// TwinCAT 3 PLC project PlcElevator
// ProgramVersion: 3.1.4024.0
// libraries:
//   Tc2_Standard, * (Beckhoff Automation GmbH)
//   Tc2_System, * (Beckhoff Automation GmbH)
//   Tc3_Module, * (Beckhoff Automation GmbH)
// project tree:
//   DUTs/ E_DoorState.TcDUT
//   GVLs/ GVL_HMI.TcGVL
//   / PlcTask.TcTTO
//   POUs/ FB_Dispatcher.TcPOU, FB_ElevatorCar.TcPOU, I_ElevatorCar.TcPOU, MAIN.TcPOU
// real-time tasks:
//   TASK PlcTask: cycle T#10ms, priority 20, ADS port 350

CONFIGURATION PlcElevator
    RESOURCE PLC ON TwinCAT3
        TASK PlcTask(INTERVAL := T#10ms, PRIORITY := 20);
        PROGRAM MAIN WITH PlcTask : MAIN;
    END_RESOURCE
END_CONFIGURATION

// ---- DUTs/E_DoorState.TcDUT
{attribute 'qualified_only'}
{attribute 'strict'}
TYPE E_DoorState :
(
	CLOSED := 0,
	OPENING := 1,
	OPEN := 2,
	CLOSING := 3
) INT;
END_TYPE

// ---- GVLs/GVL_HMI.TcGVL
{attribute 'qualified_only'}
VAR_GLOBAL
	bFloorCallsOutside : ARRAY[1..10] OF BOOL; // HMI Landing Call Buttons
	bCabinCallsInside  : ARRAY[1..10] OF BOOL; // HMI Internal Cabin Buttons
	bHmiObstruction    : BOOL;                // HMI Door Obstruction Toggle
	
	// Status Feedbacks for HMI Animation
	rfHmiCabinPosition : LREAL := 1.0;        // Continuous position (1.0 to 10.0)
	nHmiCurrentFloor   : INT := 1;            // Discrete Current Floor
	eHmiDoorState      : INT;                 // Casted E_DoorState for HMI binding
	bHmiMovingUp       : BOOL;                // Cabin is moving up
	bHmiMovingDown     : BOOL;                // Cabin is moving down
	nHmiTargetFloor    : INT;                 // Current Target Floor
END_VAR

// ---- POUs/I_ElevatorCar.TcPOU
INTERFACE I_ElevatorCar

PROPERTY CurrentFloor : INT
GET
END_GET
END_PROPERTY

PROPERTY DoorState : E_DoorState
GET
END_GET
END_PROPERTY

PROPERTY IsBusy : BOOL
GET
END_GET
END_PROPERTY

METHOD MoveToFloor : BOOL
VAR_INPUT
	nFloor : INT;
END_VAR
END_METHOD

METHOD OpenDoors : BOOL
END_METHOD

PROPERTY Position : LREAL
GET
END_GET
END_PROPERTY

END_INTERFACE

// ---- POUs/MAIN.TcPOU
PROGRAM MAIN
VAR
	fbCar : FB_ElevatorCar;
	fbDispatcher : FB_Dispatcher;

	// Automated Test Harness
	bRunTestCases : BOOL := FALSE;
	nTestStep : INT := 0;
	iTest : INT;
END_VAR

// Execute the physical elevator cabin simulation and door state machine
fbCar();

// Execute dispatcher to run SCAN sorting algorithm
fbDispatcher.Update(fbCar);

// Bind local state feedbacks to GVL_HMI for HMI animation and telemetry
GVL_HMI.rfHmiCabinPosition := fbCar.Position;
GVL_HMI.nHmiCurrentFloor   := fbCar.CurrentFloor;
GVL_HMI.eHmiDoorState      := TO_INT(fbCar.DoorState);
GVL_HMI.bHmiMovingUp       := fbDispatcher.bMovingUp;
GVL_HMI.bHmiMovingDown     := fbDispatcher.bMovingDown;
GVL_HMI.nHmiTargetFloor    := fbDispatcher.nTargetFloor;

// Automated Test Runner (Self-Verification)
IF bRunTestCases THEN
	CASE nTestStep OF
		0: // Step 0: Initialize test, clear all calls, reset cabin to floor 1
			FOR iTest := 1 TO 10 DO
				GVL_HMI.bFloorCallsOutside[iTest] := FALSE;
				GVL_HMI.bCabinCallsInside[iTest] := FALSE;
			END_FOR
			fbCar.MoveToFloor(1);
			nTestStep := 1;
			
		1: // Step 1: Wait for cabin to reach floor 1 and become idle
			IF fbCar.CurrentFloor = 1 AND NOT fbCar.IsBusy THEN
				// Place calls at floor 10 and floor 5
				GVL_HMI.bFloorCallsOutside[10] := TRUE;
				GVL_HMI.bFloorCallsOutside[5]  := TRUE;
				nTestStep := 2;
			END_IF
			
		2: // Step 2: Verify it stops at Floor 5 on the way up and clears call
			IF fbCar.CurrentFloor = 5 AND fbCar.DoorState = E_DoorState.OPEN THEN
				IF NOT GVL_HMI.bFloorCallsOutside[5] THEN
					// Floor 5 stop verified and call cleared successfully!
					nTestStep := 3;
				END_IF
			END_IF
			
		3: // Step 3: Wait for cabin to reach Floor 10 and clear call
			IF fbCar.CurrentFloor = 10 AND fbCar.DoorState = E_DoorState.OPEN THEN
				IF NOT GVL_HMI.bFloorCallsOutside[10] THEN
					// Floor 10 stop verified and call cleared successfully!
					// Test passed!
					bRunTestCases := FALSE;
					nTestStep := 0;
				END_IF
			END_IF
	END_CASE
END_IF

END_PROGRAM

// ---- POUs/FB_ElevatorCar.TcPOU
FUNCTION_BLOCK FB_ElevatorCar IMPLEMENTS I_ElevatorCar
VAR
	rfPosition : LREAL := 1.0;
	nTargetFloor : INT := 1;
	eDoorState : E_DoorState := E_DoorState.CLOSED;
	bMoving : BOOL := FALSE;
	bObstruction : BOOL := FALSE;
	bTriggerDoorOpen : BOOL := FALSE;

	fbDoorDwellTimer : TON;
	fbOpeningTimer : TON;
	fbClosingTimer : TON;
END_VAR

// Synchronize door obstruction from external HMI/safety input
bObstruction := GVL_HMI.bHmiObstruction;

// Door State Machine
CASE eDoorState OF
	E_DoorState.CLOSED:
		fbOpeningTimer(IN := FALSE);
		fbDoorDwellTimer(IN := FALSE);
		fbClosingTimer(IN := FALSE);
		
		IF bTriggerDoorOpen THEN
			bTriggerDoorOpen := FALSE;
			eDoorState := E_DoorState.OPENING;
		END_IF
		
	E_DoorState.OPENING:
		fbOpeningTimer(IN := TRUE, PT := T#1S); // 1s opening time
		IF fbOpeningTimer.Q THEN
			fbOpeningTimer(IN := FALSE);
			eDoorState := E_DoorState.OPEN;
		END_IF
		
	E_DoorState.OPEN:
		fbDoorDwellTimer(IN := NOT bObstruction, PT := T#3S); // 3s dwell timer
		IF fbDoorDwellTimer.Q THEN
			fbDoorDwellTimer(IN := FALSE);
			eDoorState := E_DoorState.CLOSING;
		END_IF
		
	E_DoorState.CLOSING:
		fbClosingTimer(IN := TRUE, PT := T#1S); // 1s closing time
		
		IF bObstruction THEN
			// Light Curtain obstruction: instantly reverse to OPENING
			fbClosingTimer(IN := FALSE);
			eDoorState := E_DoorState.OPENING;
		ELSIF fbClosingTimer.Q THEN
			fbClosingTimer(IN := FALSE);
			eDoorState := E_DoorState.CLOSED;
		END_IF
END_CASE

// Cabin Movement Logic (Safety Interlock)
IF eDoorState = E_DoorState.CLOSED THEN
	IF rfPosition < INT_TO_LREAL(nTargetFloor) THEN
		bMoving := TRUE;
		rfPosition := rfPosition + 0.02;
		IF rfPosition >= INT_TO_LREAL(nTargetFloor) THEN
			rfPosition := INT_TO_LREAL(nTargetFloor);
			bMoving := FALSE;
			bTriggerDoorOpen := TRUE; // Auto-open doors upon arrival
		END_IF
	ELSIF rfPosition > INT_TO_LREAL(nTargetFloor) THEN
		bMoving := TRUE;
		rfPosition := rfPosition - 0.02;
		IF rfPosition <= INT_TO_LREAL(nTargetFloor) THEN
			rfPosition := INT_TO_LREAL(nTargetFloor);
			bMoving := FALSE;
			bTriggerDoorOpen := TRUE; // Auto-open doors upon arrival
		END_IF
	ELSE
		bMoving := FALSE;
	END_IF
ELSE
	// Door is NOT closed - safety interlock: cabin CANNOT move
	bMoving := FALSE;
END_IF

METHOD MoveToFloor : BOOL
VAR_INPUT
	nFloor : INT;
END_VAR
IF nFloor >= 1 AND nFloor <= 10 AND eDoorState = E_DoorState.CLOSED THEN
	nTargetFloor := nFloor;
	MoveToFloor := TRUE;
ELSE
	MoveToFloor := FALSE;
END_IF
END_METHOD

METHOD OpenDoors : BOOL
IF NOT bMoving AND eDoorState = E_DoorState.CLOSED THEN
	bTriggerDoorOpen := TRUE;
	OpenDoors := TRUE;
ELSE
	OpenDoors := FALSE;
END_IF
END_METHOD

PROPERTY CurrentFloor : INT
GET
CurrentFloor := LREAL_TO_INT(rfPosition);
END_GET
END_PROPERTY

PROPERTY DoorState : E_DoorState
GET
DoorState := eDoorState;
END_GET
END_PROPERTY

PROPERTY IsBusy : BOOL
GET
IsBusy := bMoving OR (eDoorState <> E_DoorState.CLOSED);
END_GET
END_PROPERTY

PROPERTY Position : LREAL
GET
Position := rfPosition;
END_GET
END_PROPERTY

END_FUNCTION_BLOCK

// ---- POUs/FB_Dispatcher.TcPOU
FUNCTION_BLOCK FB_Dispatcher
VAR
	bMovingUp : BOOL := FALSE;
	bMovingDown : BOOL := FALSE;
	nTargetFloor : INT := 0; // 0 means no target (idle)
END_VAR

METHOD Update : BOOL
VAR_INPUT
	refCar : I_ElevatorCar;
END_VAR
VAR
	rfPos : LREAL;
	nCurrentFloor : INT;
	bHasCallsAhead : BOOL;
	bHasCallsBehind : BOOL;
	nNextTarget : INT;
	i : INT;
	bCallActive : BOOL;
END_VAR
IF refCar = 0 THEN // Null check for interface
	Update := FALSE;
	RETURN;
END_IF

rfPos := refCar.Position;
nCurrentFloor := refCar.CurrentFloor;

// 1. Clear calls on current floor if the doors are open/opening/closing
IF nTargetFloor <> 0 AND nCurrentFloor = nTargetFloor AND refCar.DoorState <> E_DoorState.CLOSED THEN
	GVL_HMI.bFloorCallsOutside[nTargetFloor] := FALSE;
	GVL_HMI.bCabinCallsInside[nTargetFloor] := FALSE;
END_IF

// 2. SCAN Algorithm State Machine
IF NOT bMovingUp AND NOT bMovingDown THEN
	// Idle State: scan for ANY call
	nNextTarget := 0;
	
	FOR i := 1 TO 10 DO
		bCallActive := GVL_HMI.bFloorCallsOutside[i] OR GVL_HMI.bCabinCallsInside[i];
		IF bCallActive THEN
			nNextTarget := i;
			EXIT; // Grab the first call we find
		END_IF
	END_FOR
	
	IF nNextTarget <> 0 THEN
		IF nNextTarget = nCurrentFloor THEN
			// Call is on current floor: just open the doors
			refCar.OpenDoors();
			GVL_HMI.bFloorCallsOutside[nNextTarget] := FALSE;
			GVL_HMI.bCabinCallsInside[nNextTarget] := FALSE;
		ELSIF nNextTarget > nCurrentFloor THEN
			bMovingUp := TRUE;
			nTargetFloor := nNextTarget;
			refCar.MoveToFloor(nTargetFloor);
		ELSE
			bMovingDown := TRUE;
			nTargetFloor := nNextTarget;
			refCar.MoveToFloor(nTargetFloor);
		END_IF
	ELSE
		nTargetFloor := 0;
	END_IF
	
ELSIF bMovingUp THEN
	// Moving Up: find nearest call ahead (above current position)
	bHasCallsAhead := FALSE;
	nNextTarget := 0;
	
	FOR i := 1 TO 10 DO
		bCallActive := GVL_HMI.bFloorCallsOutside[i] OR GVL_HMI.bCabinCallsInside[i];
		IF bCallActive AND INT_TO_LREAL(i) > (rfPos - 0.05) THEN
			IF NOT bHasCallsAhead OR i < nNextTarget THEN
				bHasCallsAhead := TRUE;
				nNextTarget := i;
			END_IF
		END_IF
	END_FOR
	
	IF bHasCallsAhead THEN
		// We have calls ahead in the Up direction: head to the nearest one
		nTargetFloor := nNextTarget;
		refCar.MoveToFloor(nTargetFloor);
	ELSE
		// No calls ahead: check if there are calls behind/below us
		bHasCallsBehind := FALSE;
		nNextTarget := 0;
		
		FOR i := 1 TO 10 DO
			bCallActive := GVL_HMI.bFloorCallsOutside[i] OR GVL_HMI.bCabinCallsInside[i];
			IF bCallActive AND INT_TO_LREAL(i) < (rfPos + 0.05) THEN
				IF NOT bHasCallsBehind OR i > nNextTarget THEN // For Down, grab highest floor first
					bHasCallsBehind := TRUE;
					nNextTarget := i;
				END_IF
			END_IF
		END_FOR
		
		IF bHasCallsBehind THEN
			// Switch direction to Down
			bMovingUp := FALSE;
			bMovingDown := TRUE;
			nTargetFloor := nNextTarget;
			refCar.MoveToFloor(nTargetFloor);
		ELSE
			// No calls at all: go idle
			bMovingUp := FALSE;
			nTargetFloor := 0;
		END_IF
	END_IF
	
ELSIF bMovingDown THEN
	// Moving Down: find nearest call ahead (below current position)
	bHasCallsAhead := FALSE;
	nNextTarget := 0;
	
	FOR i := 1 TO 10 DO
		bCallActive := GVL_HMI.bFloorCallsOutside[i] OR GVL_HMI.bCabinCallsInside[i];
		IF bCallActive AND INT_TO_LREAL(i) < (rfPos + 0.05) THEN
			IF NOT bHasCallsAhead OR i > nNextTarget THEN
				bHasCallsAhead := TRUE;
				nNextTarget := i;
			END_IF
		END_IF
	END_FOR
	
	IF bHasCallsAhead THEN
		// We have calls ahead in the Down direction: head to the nearest one
		nTargetFloor := nNextTarget;
		refCar.MoveToFloor(nTargetFloor);
	ELSE
		// No calls ahead: check if there are calls behind/above us
		bHasCallsBehind := FALSE;
		nNextTarget := 0;
		
		FOR i := 1 TO 10 DO
			bCallActive := GVL_HMI.bFloorCallsOutside[i] OR GVL_HMI.bCabinCallsInside[i];
			IF bCallActive AND INT_TO_LREAL(i) > (rfPos - 0.05) THEN
				IF NOT bHasCallsBehind OR i < nNextTarget THEN // For Up, grab lowest floor first
					bHasCallsBehind := TRUE;
					nNextTarget := i;
				END_IF
			END_IF
		END_FOR
		
		IF bHasCallsBehind THEN
			// Switch direction to Up
			bMovingDown := FALSE;
			bMovingUp := TRUE;
			nTargetFloor := nNextTarget;
			refCar.MoveToFloor(nTargetFloor);
		ELSE
			// No calls at all: go idle
			bMovingDown := FALSE;
			nTargetFloor := 0;
		END_IF
	END_IF
END_IF

Update := TRUE;
END_METHOD

END_FUNCTION_BLOCK
